// SIMATIC S7-200 SMART project (STEP 7-Micro/WIN SMART), CPU ST40

ORGANIZATION_BLOCK MAIN:OB1
TITLE=程序注释    跑马灯共含有8个灯
BEGIN
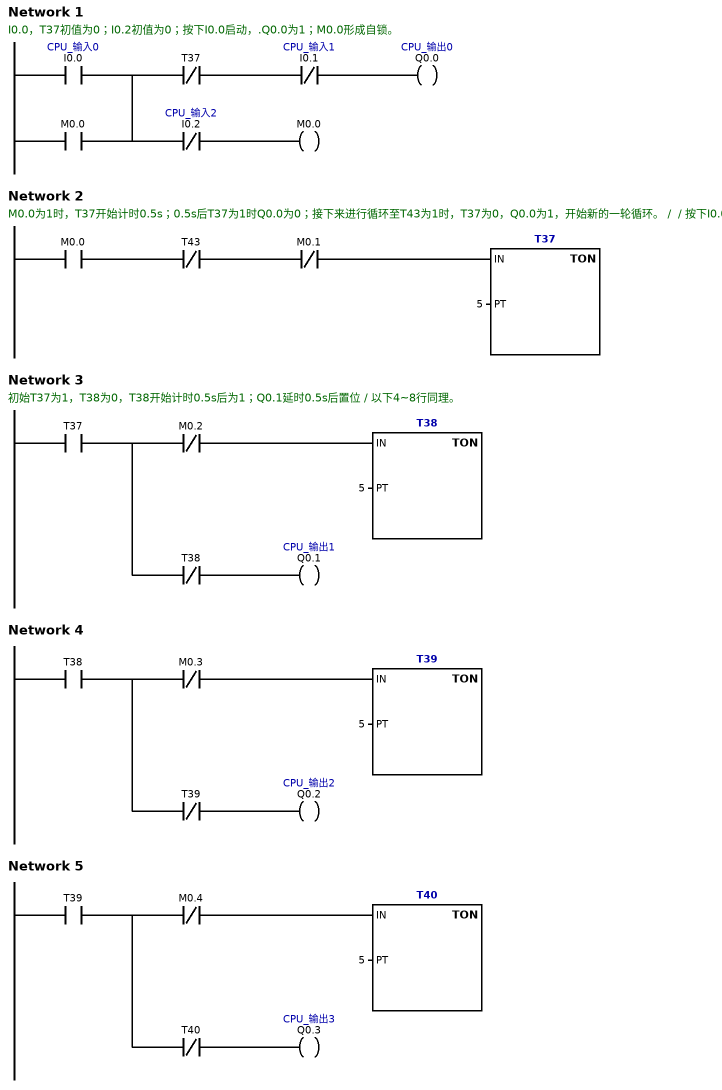
Network 1
// I0.0，T37初值为0；I0.2初值为0；按下I0.0启动，.Q0.0为1；M0.0形成自锁。
LD     CPU_输入0:I0.0
O      M0.0
LPS
AN     T37
AN     CPU_输入1:I0.1
=      CPU_输出0:Q0.0
LPP
AN     CPU_输入2:I0.2
=      M0.0
Network 2
// M0.0为1时，T37开始计时0.5s；0.5s后T37为1时Q0.0为0；接下来进行循环至T43为1时，T37为0，Q0.0为1，开始新的一轮循环。
// 
// 按下I0.0T37开始计时0.5s，计时0.5s后T37为1。
LD     M0.0
AN     T43
AN     M0.1
TON    T37, 5
Network 3
// 初始T37为1，T38为0，T38开始计时0.5s后为1；Q0.1延时0.5s后置位
// 以下4~8行同理。
LD     T37
LPS
AN     M0.2
TON    T38, 5
LPP
AN     T38
=      CPU_输出1:Q0.1
Network 4
LD     T38
LPS
AN     M0.3
TON    T39, 5
LPP
AN     T39
=      CPU_输出2:Q0.2
Network 5
LD     T39
LPS
AN     M0.4
TON    T40, 5
LPP
AN     T40
=      CPU_输出3:Q0.3
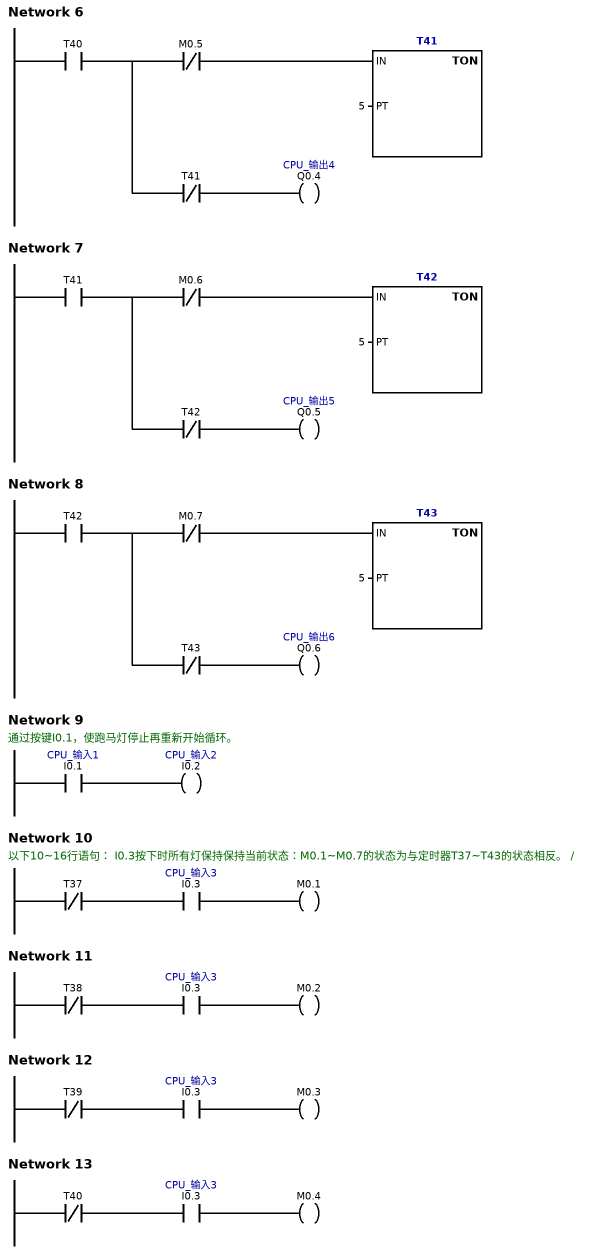
Network 6
LD     T40
LPS
AN     M0.5
TON    T41, 5
LPP
AN     T41
=      CPU_输出4:Q0.4
Network 7
LD     T41
LPS
AN     M0.6
TON    T42, 5
LPP
AN     T42
=      CPU_输出5:Q0.5
Network 8
LD     T42
LPS
AN     M0.7
TON    T43, 5
LPP
AN     T43
=      CPU_输出6:Q0.6
Network 9
// 通过按键I0.1，使跑马灯停止再重新开始循环。
LD     CPU_输入1:I0.1
=      CPU_输入2:I0.2
Network 10
// 以下10~16行语句： I0.3按下时所有灯保持保持当前状态：M0.1~M0.7的状态为与定时器T37~T43的状态相反。
// 
LDN    T37
A      CPU_输入3:I0.3
=      M0.1
Network 11
LDN    T38
A      CPU_输入3:I0.3
=      M0.2
Network 12
LDN    T39
A      CPU_输入3:I0.3
=      M0.3
Network 13
LDN    T40
A      CPU_输入3:I0.3
=      M0.4
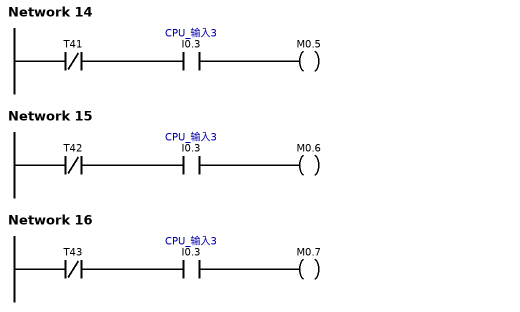
Network 14
LDN    T41
A      CPU_输入3:I0.3
=      M0.5
Network 15
LDN    T42
A      CPU_输入3:I0.3
=      M0.6
Network 16
LDN    T43
A      CPU_输入3:I0.3
=      M0.7
END_ORGANIZATION_BLOCK
